{attribute 'linkalways'} 
{attribute 'no_explicit_call' := 'This FB is a CLASS and must be accessed using methods or properties'}
{attribute 'enable_dynamic_creation'}
FUNCTION_BLOCK MissingNodePrototypeDeserializationError EXTENDS Error
VAR
	nodeType : T_MAXSTRING;
END_VAR

PROPERTY PUBLIC ErrorType : T_MAXSTRING
GET
ErrorType := 'MISSING_NODE_PROTOTYPE_DESERIALIZATION_ERROR';
END_GET
END_PROPERTY

METHOD FB_init : BOOL
VAR_INPUT
	bInitRetains : BOOL; // if TRUE, the retain variables are initialized (warm start / cold start)
	bInCopyCode : BOOL;  // if TRUE, the instance afterwards gets moved into the copy code (online change)
	MissingType : T_MAXSTRING;
END_VAR
 nodeType := MissingType;
END_METHOD

PROPERTY PUBLIC Message : T_MAXSTRING
GET
Message := CONCAT('Deserialization Failed, Missing Node Prototype : ',nodeType);
END_GET
END_PROPERTY

END_FUNCTION_BLOCK

(* stored: Version 1.1.0.1, ProductVersion 3.1.4024.12
   POU MissingNodePrototypeDeserializationError: Id {3c97932d-0312-4719-9024-3d6e6859f592}, SpecialFunc None
   Folder Constructor: Id {9a6ecff5-b807-4505-b997-e5486b1e04f0}
   Property ErrorType: Id {64f7e5c8-04aa-4911-b08c-8065a204dacf}
   Get Get: Id {33b7c5ee-7b5d-44d4-9895-6e788ada1aba}
   Method FB_init: Id {00fdec9d-0922-46c3-a790-471354ed631e}
   Property Message: Id {eb05180d-8f15-4349-9789-a9d690e6ed9d}
   Get Get: Id {81abb13d-8b5f-428f-aed9-84fb87053b4a} *)
